FUNCTION Convert_REAL_TO_USINT : Hresult
VAR_INPUT
	in : REAL;
	out : REFERENCE TO USINT;
END_VAR
VAR
	converted : USINT;
END_VAR

converted := REAL_TO_USINT(in);

IF (USINT_TO_REAL(converted) <> in) THEN
	Convert_REAL_TO_USINT := INCOMPATIBLE;
	RETURN;
END_IF

out := converted;

END_FUNCTION

(* stored: Version 1.1.0.1, ProductVersion 3.1.4024.12
   POU Convert_REAL_TO_USINT: Id {4fb984c6-8c9d-4864-8fb2-afdd84fbf27b}, SpecialFunc None *)
